{attribute addProperty BoxType "AT2025-0250-0023"}
{attribute addProperty Id "A_0076_AT2001_5250_0017_AT2001_5250AT2001_3DCFC8D064080"}
{attribute addProperty CRC "684300042"}
{attribute addProperty SizeInBites "640"}
{attribute addProperty SizeInBytes "80"}
TYPE A_0064_AT2025_0250_0023_AT2025_0250_28C9970A EXTENDS AT2025_9506A482 :
STRUCT
	{attribute addProperty Name "A_0076_AT2001_5250_0017_AT2001_5250"}
	A_0076_AT2001_5250_0017_AT2001_5250 : AT2001_3DCFC8D0;
END_STRUCT
END_TYPE

(* stored: Version 1.2.0.0, ProductVersion 3.1.4024.9
   DUT A_0064_AT2025_0250_0023_AT2025_0250_28C9970A: Id {cee26e5e-998a-4a31-903a-c962b596ba44} *)
